(* IEC 61131-3 sources: volt/packages/volt-lsp-iec/test-corpus/lenze-mid/Device/Plc Logic/Application/Library Manager/SysProcess Implementation, 12 files *)

(* ---- SYSPROCESSCREATE.pou ---- *)
FUNCTION SYSPROCESSCREATE : RTS_IEC_HANDLE
VAR_INPUT
	PSZAPPLICATION : REFERENCE TO STRING;
	PSZCOMMANDLINE : REFERENCE TO STRING;
	ULHIDE : UDINT;
	PRESULT : POINTER TO RTS_IEC_RESULT;
END_VAR
END_FUNCTION

(* ---- SYSPROCESSCREATE2.pou ---- *)
FUNCTION SYSPROCESSCREATE2 : RTS_IEC_HANDLE
VAR_INPUT
	PSZAPPLICATION : REFERENCE TO STRING;
	PSZCOMMANDLINE : REFERENCE TO STRING;
	ULFLAGS : UDINT;
	PRESULT : POINTER TO RTS_IEC_RESULT;
END_VAR
END_FUNCTION

(* ---- SYSPROCESSEXECUTECOMMAND.pou ---- *)
FUNCTION SYSPROCESSEXECUTECOMMAND : DINT
VAR_INPUT
	PSZCOMAND : REFERENCE TO STRING;
	PRESULT : POINTER TO RTS_IEC_RESULT;
END_VAR
END_FUNCTION

(* ---- SYSPROCESSEXECUTECOMMAND2.pou ---- *)
FUNCTION SYSPROCESSEXECUTECOMMAND2 : DINT
VAR_INPUT
	PSZCOMMAND : REFERENCE TO STRING;
	PSZSTDOUT : REFERENCE TO STRING;
	UDISTDOUTLEN : UDINT;
	PRESULT : POINTER TO RTS_IEC_RESULT;
END_VAR
END_FUNCTION

(* ---- SYSPROCESSFREEHANDLE.pou ---- *)
FUNCTION SYSPROCESSFREEHANDLE : RTS_IEC_RESULT
VAR_INPUT
	HPROCESS : RTS_IEC_HANDLE;
END_VAR
END_FUNCTION

(* ---- SYSPROCESSGETCURRENTHANDLE.pou ---- *)
FUNCTION SYSPROCESSGETCURRENTHANDLE : RTS_IEC_HANDLE
VAR_INPUT
	PRESULT : POINTER TO RTS_IEC_RESULT;
END_VAR
END_FUNCTION

(* ---- SYSPROCESSGETOSID.pou ---- *)
FUNCTION SYSPROCESSGETOSID : UDINT
VAR_INPUT
	HPROCESS : RTS_IEC_HANDLE;
	PRESULT : POINTER TO RTS_IEC_RESULT;
END_VAR
END_FUNCTION

(* ---- SYSPROCESSGETPRIORITY.pou ---- *)
FUNCTION SYSPROCESSGETPRIORITY : RTS_IEC_RESULT
VAR_INPUT
	HPROCESS : RTS_IEC_HANDLE;
	PULPRIORITY : POINTER TO UDINT;
END_VAR
END_FUNCTION

(* ---- SYSPROCESSGETSTATE.pou ---- *)
FUNCTION SYSPROCESSGETSTATE : RTS_IEC_RESULT
VAR_INPUT
	HPROCESS : RTS_IEC_HANDLE;
	PULSTATE : POINTER TO UDINT;
END_VAR
END_FUNCTION

(* ---- SYSPROCESSRESUME.pou ---- *)
FUNCTION SYSPROCESSRESUME : RTS_IEC_RESULT
VAR_INPUT
	HPROCESS : RTS_IEC_HANDLE;
END_VAR
END_FUNCTION

(* ---- SYSPROCESSSETPRIORITY.pou ---- *)
FUNCTION SYSPROCESSSETPRIORITY : RTS_IEC_RESULT
VAR_INPUT
	HPROCESS : RTS_IEC_HANDLE;
	ULPRIORITY : UDINT;
END_VAR
END_FUNCTION

(* ---- SYSPROCESSTERMINATE.pou ---- *)
FUNCTION SYSPROCESSTERMINATE : RTS_IEC_RESULT
VAR_INPUT
	HPROCESS : RTS_IEC_HANDLE;
END_VAR
END_FUNCTION
